PROGRAM idle
VAR
	ed_routine_idle: BOOL;
	redox_doser_idle_enable: BOOL;
	
	tmr_idle_pumps: TON;
	u_3112_a_idle_request: BOOL;
	u_3312_a_idle_request: BOOL;
	u_3405_a_idle_request: BOOL;
	u_3212_a_idle_request: BOOL;
	tmr_idle_pump_delay: TON;
	u_3112_a_running: BOOL;
	u_3112_a_speed_ref: INT;
	u_3112_a_sp: REAL;
	salt_pressure_actual: REAL;
	u_3112_a_ready: BOOL;
	u_3212_a_running: BOOL;
	u_3212_a_ready: BOOL;
	u_3312_a_ready: BOOL;
	u_3312_a_running: BOOL;
	u_3405_a_running: BOOL;
	u_3405_a_ready: BOOL;
	stack_power_enable: BOOL;
	nv_3110_a_open_request: BOOL;
	nv_3210_a_open_request: BOOL;
	nv_3310_a_open_request: BOOL;
	nv_3110_a_open_feedback: BOOL;
	nv_3210_a_open_feedback: BOOL;
	nv_3310_a_open_feedback: BOOL;
	nv_3110_a_idle_request: BOOL;
	nv_3210_a_idle_request: BOOL;
	nv_3310_a_idle_request: BOOL;
	nv_3135_a_idle_request: BOOL;
	nv_3235_a_idle_request: BOOL;
	nv_3335_a_idle_request: BOOL;
	nv_3372_a_idle_request: BOOL;
	nv_3162_a_idle_request: BOOL;

	idle_stack_power_enable: BOOL;
	idle_TEMP_BIT: BOOL;
	tmr_idle_valye_delay: TON;
	tmr_idle_valve_delay: TON;
	tmr_idle_valve_delay_et: TIME;
	tmr_idle_valve_delay_pt: TIME := T#20S;
	tmr_idle_valve_delay_q: BOOL;
	u_3112_a_idle_pressure_setpoint_request: REAL;
	u_3212_a_idle_pressure_setpoint_request: REAL;
	u_3312_a_idle_pressure_setpoint_request: REAL;
	u_3405_a_idle_pressure_setpoint_request: REAL;
	idle_stable: BOOL;
	av_3148_a_idle_position_request: REAL;
	av_3248_a_idle_position_request: REAL;
	av_3348_a_idle_position_request: REAL;
	redox_pressure_calculation: REAL;
	redox_idle_pressure_sp_request: REAL;
	idle_startup_ons: R_TRIG;
END_VAR
VAR // added by the converter: edge detectors and wires of the graphical bodies
    _w1, _w2, _w3, _w4 : BOOL;
END_VAR

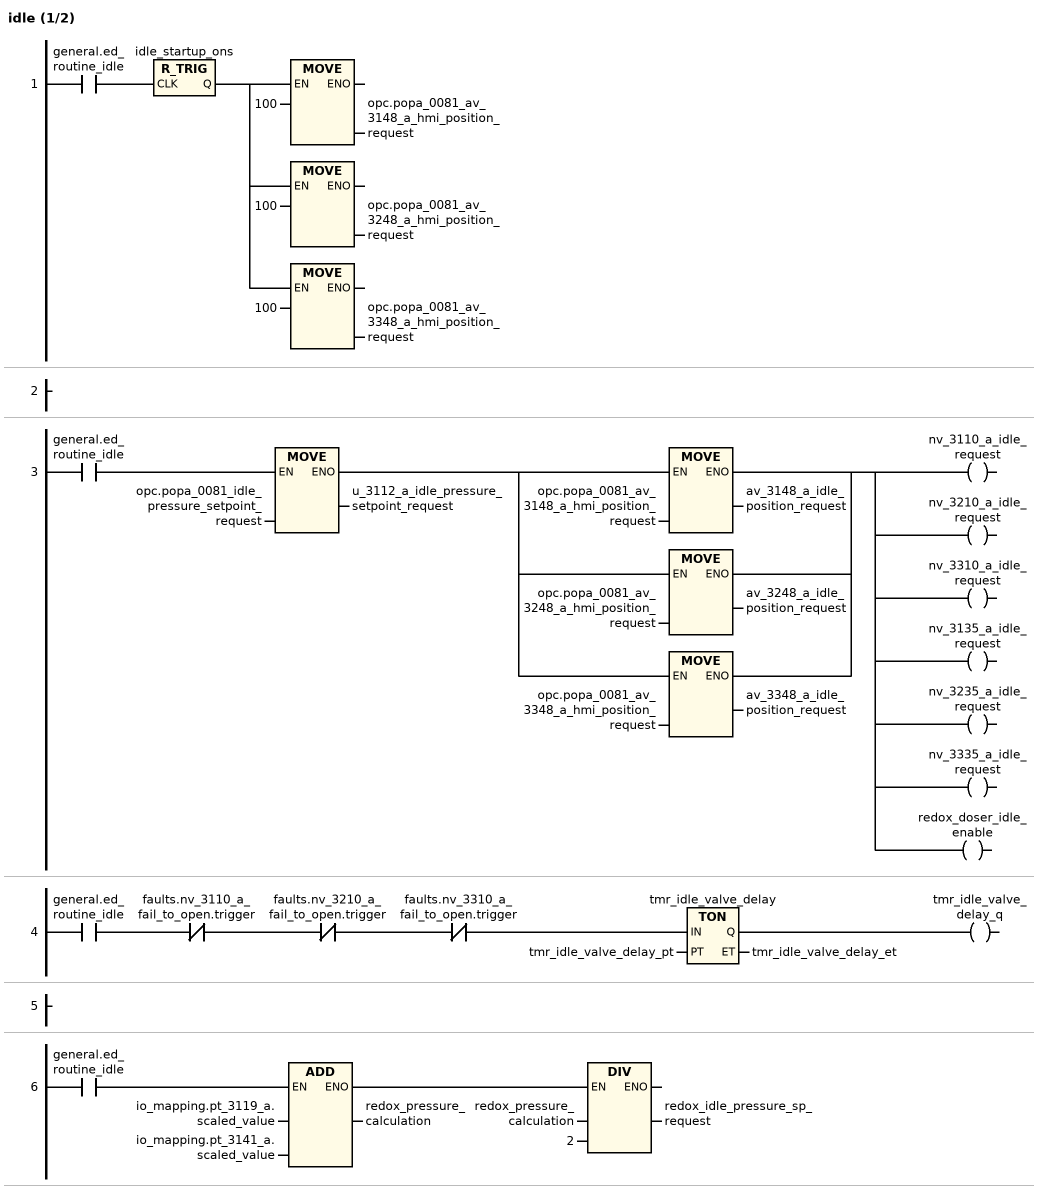
// NETWORK 1
idle_startup_ons(CLK := general.ed_routine_idle); // R_TRIG
IF idle_startup_ons.Q THEN opc.popa_0081_av_3148_a_hmi_position_request := 100; END_IF
IF idle_startup_ons.Q THEN opc.popa_0081_av_3248_a_hmi_position_request := 100; END_IF
IF idle_startup_ons.Q THEN opc.popa_0081_av_3348_a_hmi_position_request := 100; END_IF

// NETWORK 2

// NETWORK 3
_w1 := general.ed_routine_idle;
IF _w1 THEN u_3112_a_idle_pressure_setpoint_request := opc.popa_0081_idle_pressure_setpoint_request; END_IF
IF _w1 THEN av_3148_a_idle_position_request := opc.popa_0081_av_3148_a_hmi_position_request; END_IF
IF _w1 THEN av_3248_a_idle_position_request := opc.popa_0081_av_3248_a_hmi_position_request; END_IF
IF _w1 THEN av_3348_a_idle_position_request := opc.popa_0081_av_3348_a_hmi_position_request; END_IF
_w2 := _w1 OR (_w1 OR _w1);
nv_3110_a_idle_request := _w2;
nv_3210_a_idle_request := _w2;
nv_3310_a_idle_request := _w2;
nv_3135_a_idle_request := _w2;
nv_3235_a_idle_request := _w2;
nv_3335_a_idle_request := _w2;
redox_doser_idle_enable := _w2;

// NETWORK 4
tmr_idle_valve_delay(
    IN := general.ed_routine_idle AND NOT faults.nv_3110_a_fail_to_open.trigger AND NOT faults.nv_3210_a_fail_to_open.trigger AND NOT faults.nv_3310_a_fail_to_open.trigger,
    PT := tmr_idle_valve_delay_pt,
    ET => tmr_idle_valve_delay_et); // TON
tmr_idle_valve_delay_q := tmr_idle_valve_delay.Q;

// NETWORK 5

// NETWORK 6
_w3 := general.ed_routine_idle;
IF _w3 THEN
    redox_pressure_calculation := io_mapping.pt_3119_a.scaled_value + io_mapping.pt_3141_a.scaled_value;
END_IF
IF _w3 THEN redox_idle_pressure_sp_request := redox_pressure_calculation / 2; END_IF

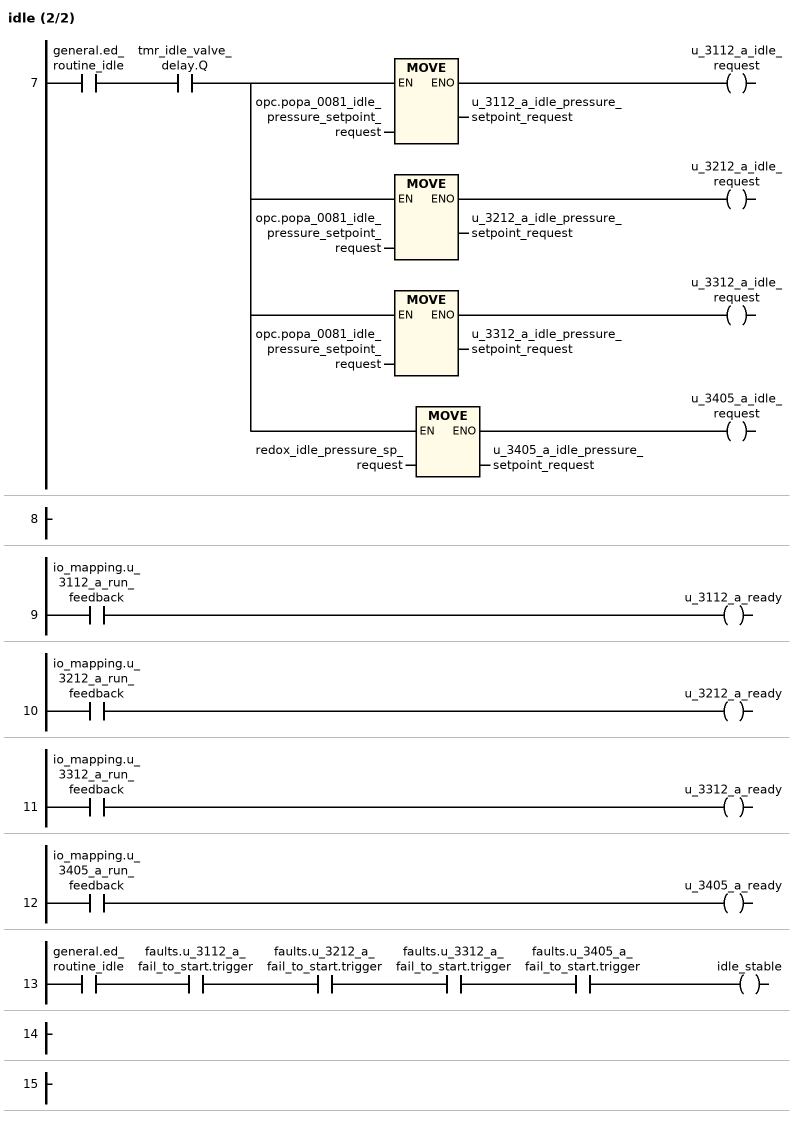
// NETWORK 7
_w4 := general.ed_routine_idle AND tmr_idle_valve_delay.Q;
IF _w4 THEN u_3112_a_idle_pressure_setpoint_request := opc.popa_0081_idle_pressure_setpoint_request; END_IF
u_3112_a_idle_request := _w4;
IF _w4 THEN u_3212_a_idle_pressure_setpoint_request := opc.popa_0081_idle_pressure_setpoint_request; END_IF
u_3212_a_idle_request := _w4;
IF _w4 THEN u_3312_a_idle_pressure_setpoint_request := opc.popa_0081_idle_pressure_setpoint_request; END_IF
u_3312_a_idle_request := _w4;
IF _w4 THEN u_3405_a_idle_pressure_setpoint_request := redox_idle_pressure_sp_request; END_IF
u_3405_a_idle_request := _w4;

// NETWORK 8

// NETWORK 9
u_3112_a_ready := io_mapping.u_3112_a_run_feedback;

// NETWORK 10
u_3212_a_ready := io_mapping.u_3212_a_run_feedback;

// NETWORK 11
u_3312_a_ready := io_mapping.u_3312_a_run_feedback;

// NETWORK 12
u_3405_a_ready := io_mapping.u_3405_a_run_feedback;

// NETWORK 13
idle_stable := general.ed_routine_idle AND faults.u_3112_a_fail_to_start.trigger AND faults.u_3212_a_fail_to_start.trigger AND faults.u_3312_a_fail_to_start.trigger AND faults.u_3405_a_fail_to_start.trigger;

// NETWORK 14

// NETWORK 15

END_PROGRAM

(* stored: Version 1.1.0.1, ProductVersion 3.1.4024.15
   POU idle: Id {3d08b1fd-a23f-437d-8121-cefd84a9c392}, SpecialFunc None *)
